Fanuc KAREL source: kt00224.KL

-- PROVISIONAL review KL for V770-1; original PC SHA256 cc69ab9f0fa94f29c4b89f0a9e8eab832f7277ed535c0188754bec09545eaa79
-- Incomplete behavior may be omitted. Consult companion uncertainty JSON. Do not deploy.
PROGRAM KT00224
%NOLOCKGROUP
VAR
  OUT : INTEGER
-- UNRESOLVED_DECL H1 type=002017
-- UNRESOLVED_DECL H2 type=002017
BEGIN
  -- UNRESOLVED_PC offsets 5-19; opcodes 2E,22,9D,33,B4
  -- UNRESOLVED_PC offsets 24-38; opcodes 2E,22,9D,33,B4
  -- UNRESOLVED_PC offsets 43-57; opcodes 2E,22,9D,33,B4
  -- UNRESOLVED_PC offsets 62-76; opcodes 2E,22,9D,33,B4
  -- UNRESOLVED_PC offsets 81-106; opcodes 22,9D,33,B3,22,9D,33,B3,46,23
  -- UNRESOLVED_PC offsets 111-115; opcodes 7F
END KT00224
